// Mitsubishi GX Works2 project: 생자 금속 단속동작   PLC: Q02/Q02H

PROGRAM MAIN
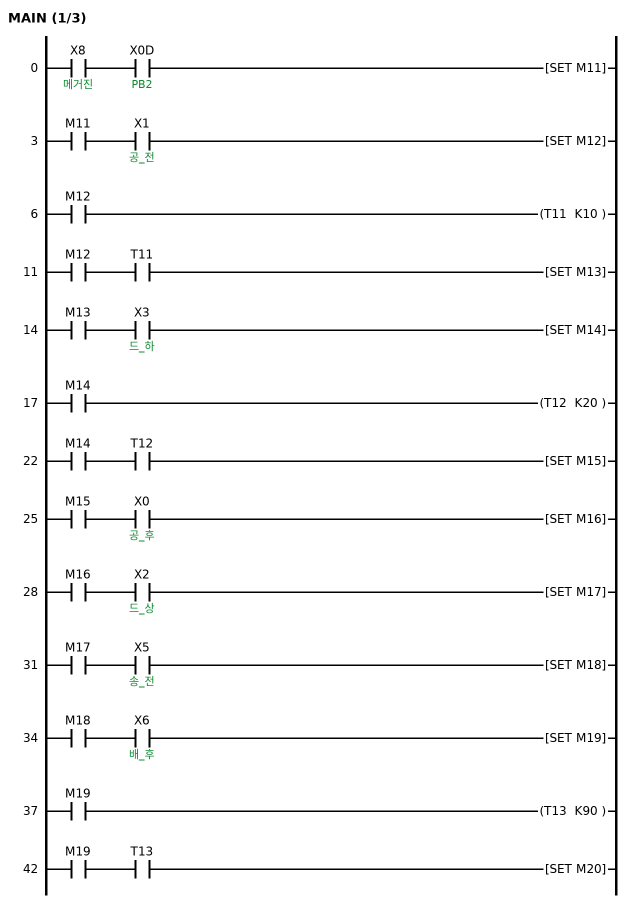
0     LD      X8  ; 메거진
      AND     X0D  ; PB2
      SET     M11
3     LD      M11
      AND     X1  ; 공_전
      SET     M12
6     LD      M12
      OUT     T11 K10
11    LD      M12
      AND     T11
      SET     M13
14    LD      M13
      AND     X3  ; 드_하
      SET     M14
17    LD      M14
      OUT     T12 K20
22    LD      M14
      AND     T12
      SET     M15
25    LD      M15
      AND     X0  ; 공_후
      SET     M16
28    LD      M16
      AND     X2  ; 드_상
      SET     M17
31    LD      M17
      AND     X5  ; 송_전
      SET     M18
34    LD      M18
      AND     X6  ; 배_후
      SET     M19
37    LD      M19
      OUT     T13 K90
42    LD      M19
      AND     T13
      SET     M20
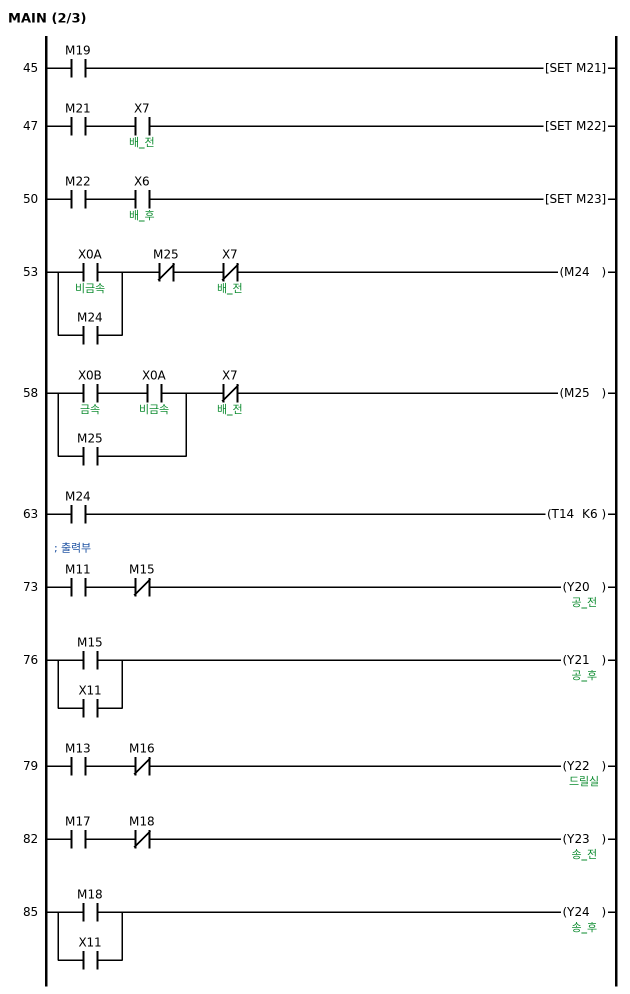
45    LD      M19
      SET     M21
47    LD      M21
      AND     X7  ; 배_전
      SET     M22
50    LD      M22
      AND     X6  ; 배_후
      SET     M23
53    LD      X0A  ; 비금속
      OR      M24
      ANI     M25
      ANI     X7  ; 배_전
      OUT     M24
58    LD      X0B  ; 금속
      AND     X0A  ; 비금속
      OR      M25
      ANI     X7  ; 배_전
      OUT     M25
63    LD      M24
      OUT     T14 K6
; 출력부
73    LD      M11
      ANI     M15
      OUT     Y20  ; 공_전
76    LD      M15
      OR      X11
      OUT     Y21  ; 공_후
79    LD      M13
      ANI     M16
      OUT     Y22  ; 드릴실
82    LD      M17
      ANI     M18
      OUT     Y23  ; 송_전
85    LD      M18
      OR      X11
      OUT     Y24  ; 송_후
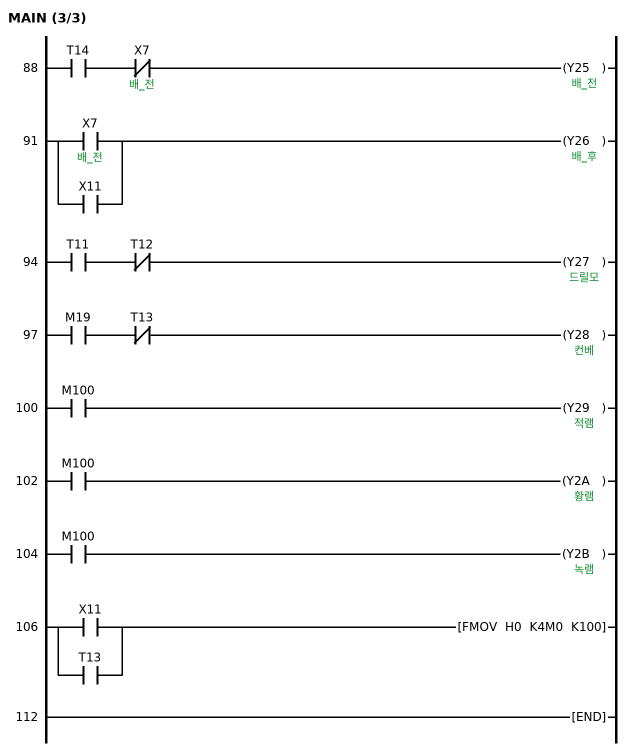
88    LD      T14
      ANI     X7  ; 배_전
      OUT     Y25  ; 배_전
91    LD      X7  ; 배_전
      OR      X11
      OUT     Y26  ; 배_후
94    LD      T11
      ANI     T12
      OUT     Y27  ; 드릴모
97    LD      M19
      ANI     T13
      OUT     Y28  ; 컨베
100   LD      M100
      OUT     Y29  ; 적램
102   LD      M100
      OUT     Y2A  ; 황램
104   LD      M100
      OUT     Y2B  ; 녹램
106   LD      X11
      OR      T13
      FMOV    H0 K4M0 K100
112   END
END_PROGRAM

// device comments not shown above
X4  ; 송_후
X9  ; 이송감지
X0C  ; PB1
X0E  ; PB3
X0F  ; 비상정지
